(* CoDeSys 2.3.9.36 project: gittest.pro *)
(* Libraries: SysLibTargetVisu.lib 7.7.04 09:17:22, STANDARD.LIB 7.7.04 09:17:22, SYSLIBCALLBACK.LIB 24.9.04 09:58:24 *)

(* POU PLC_PRG, ST *)
PROGRAM PLC_PRG
VAR
	x	: INT;

END_VAR
x := 1;
END_PROGRAM
